{attribute 'qualified_only'}
VAR_GLOBAL
	
	sensorN1 AT %I* : BOOL ;
	sensorN2 AT %I* : BOOL ;
	
	valveN1 AT %Q* : BOOL;
	ValveN2 AT %Q* : BOOL;
	
	bStartMeasurement : BOOL := FALSE;
	
	
END_VAR

(* stored: Version 1.1.0.1, ProductVersion 3.1.4024.13
   GVL GVL: Id {e2b737e1-ecfa-4c3d-8282-12247fb57bf5} *)
